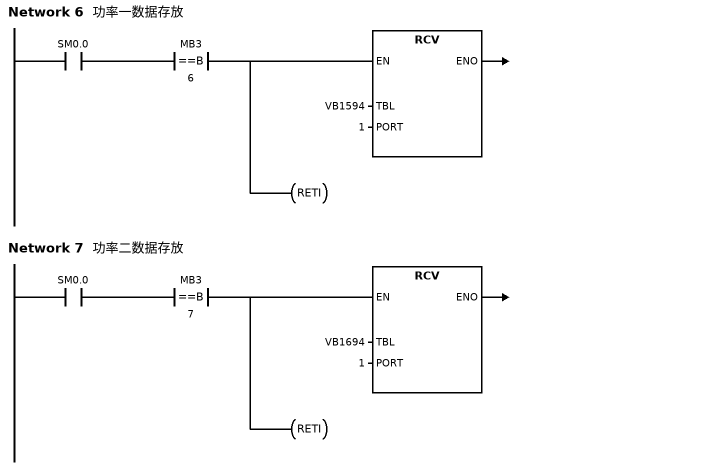
[picture p24: INT0 networks 6-7]
Network 6 // 功率一数据存放
LD     SM0.0
AB=    MB3, 6
RCV    VB1594, 1
CRETI
Network 7 // 功率二数据存放
LD     SM0.0
AB=    MB3, 7
RCV    VB1694, 1
CRETI
END_INTERRUPT_BLOCK

INTERRUPT_BLOCK 高速采集压力:INT1
TITLE=中断例行程序注解
BEGIN
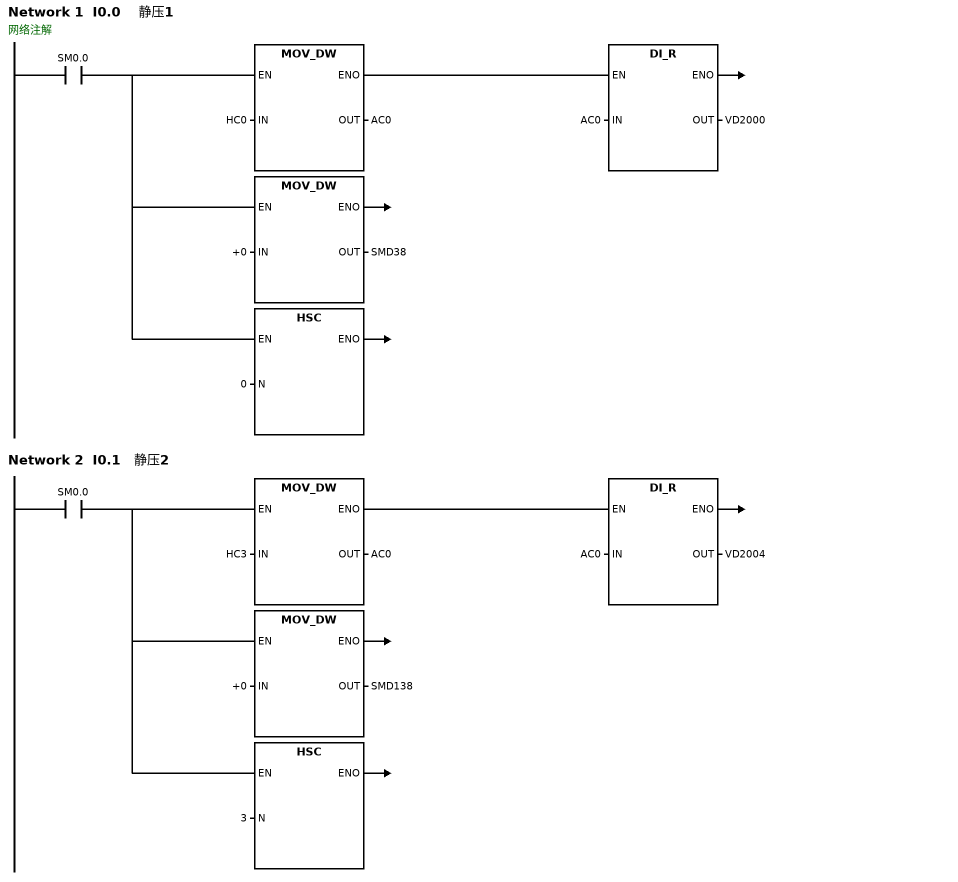
Network 1 // I0.0    静压1
// 网络注解
LD     SM0.0
LPS
MOVD   HC0, AC0
AENO
DTR    AC0, VD2000
LRD
MOVD   +0, SMD38
LPP
HSC    0
Network 2 // I0.1   静压2
LD     SM0.0
LPS
MOVD   HC3, AC0
AENO
DTR    AC0, VD2004
LRD
MOVD   +0, SMD138
LPP
HSC    3
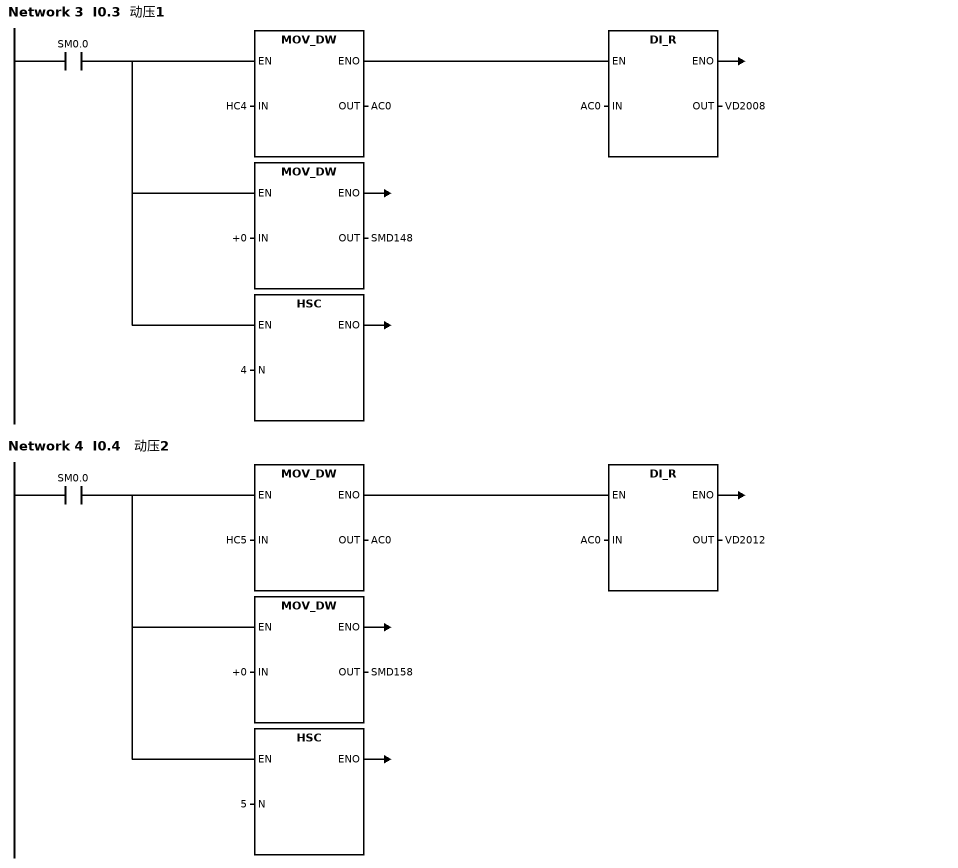
Network 3 // I0.3  动压1
LD     SM0.0
LPS
MOVD   HC4, AC0
AENO
DTR    AC0, VD2008
LRD
MOVD   +0, SMD148
LPP
HSC    4
Network 4 // I0.4   动压2
LD     SM0.0
LPS
MOVD   HC5, AC0
AENO
DTR    AC0, VD2012
LRD
MOVD   +0, SMD158
LPP
HSC    5
Network 11 // 网络标题
// 网络注释
Network 17 // 网络标题
// 网络注释
END_INTERRUPT_BLOCK
